SEGMENT_TYPE EIP (* EIP Segment *)
  (* Standard: 61499 ITA; Description: EIP ... *)
  (* Version 0.1, 2008-07-03, tstras, Profactor GmbH *)
  (* Compiler header: abc.xyz *)
  (* Compiler classdef: EIP .... *)
  (* Compiler Java IBM VisualAge 3.0 *)
  VAR_INPUT
    Param : WSTRING; (* Param *)
  END_VAR
END_SEGMENT_TYPE
